KUKA KRL program: Reset_CT.src, Reset_CT.dat

--- Reset_CT.src ---
&ACCESS RVP
&REL 1
DEF  Reset_CT ( )
   ;FOLD INI;%{PE}
      ;FOLD BASISTECH INI
         GLOBAL INTERRUPT DECL 3 WHEN $STOPMESS==TRUE DO IR_STOPM ( )
         INTERRUPT ON 3
         BAS (#INITMOV,0 )
      ;ENDFOLD (BASISTECH INI)
      ;FOLD USER INI
         ;Make your modifications here

      ;ENDFOLD (USER INI)
   ;ENDFOLD (INI)

;Pone a 0 contadore de tiempo de ciclo

;Control Tiempo de ciclo
ALT_TC=1
POS_BAT_TC=1
INDICE_RACK=1
INDICE_PICK=1
INDICE_DROP=1
INDICE_ARRAYS_CPB=1
INDICE_ARRAYS_CPS=1

TC_PICK_RACK1[1]=0
TC_PICK_RACK1[2]=0
TC_PICK_RACK1[3]=0
TC_PICK_RACK1[4]=0
TC_PICK_RACK1[5]=0
TC_PICK_RACK1[6]=0
TC_PICK_RACK1[7]=0
TC_PICK_RACK1[8]=0
TC_PICK_RACK1[9]=0
TC_PICK_RACK1[10]=0
TC_PICK_RACK1[11]=0
TC_PICK_RACK1[12]=0
TC_PICK_RACK1[13]=0
TC_PICK_RACK1[14]=0
TC_PICK_RACK1[15]=0
TC_PICK_RACK1[16]=0
TC_PICK_RACK1[17]=0
TC_PICK_RACK1[18]=0
TC_PICK_RACK1[19]=0
TC_PICK_RACK1[20]=0
TC_PICK_RACK1[21]=0
TC_PICK_RACK1[22]=0
TC_PICK_RACK1[23]=0
TC_PICK_RACK1[24]=0
TC_PICK_RACK1[25]=0
TC_PICK_RACK1[26]=0
TC_PICK_RACK1[27]=0
TC_PICK_RACK1[28]=0
TC_PICK_RACK1[29]=0
TC_PICK_RACK1[30]=0
TC_PICK_RACK1[31]=0
TC_PICK_RACK1[32]=0
TC_PICK_RACK1[33]=0
TC_PICK_RACK1[34]=0
TC_PICK_RACK1[35]=0
TC_PICK_RACK1[36]=0

TC_PICK_RACK2[1]=0
TC_PICK_RACK2[2]=0
TC_PICK_RACK2[3]=0
TC_PICK_RACK2[4]=0
TC_PICK_RACK2[5]=0
TC_PICK_RACK2[6]=0
TC_PICK_RACK2[7]=0
TC_PICK_RACK2[8]=0
TC_PICK_RACK2[9]=0
TC_PICK_RACK2[10]=0
TC_PICK_RACK2[11]=0
TC_PICK_RACK2[12]=0
TC_PICK_RACK2[13]=0
TC_PICK_RACK2[14]=0
TC_PICK_RACK2[15]=0
TC_PICK_RACK2[16]=0
TC_PICK_RACK2[17]=0
TC_PICK_RACK2[18]=0
TC_PICK_RACK2[19]=0
TC_PICK_RACK2[20]=0
TC_PICK_RACK2[21]=0
TC_PICK_RACK2[22]=0
TC_PICK_RACK2[23]=0
TC_PICK_RACK2[24]=0
TC_PICK_RACK2[25]=0
TC_PICK_RACK2[26]=0
TC_PICK_RACK2[27]=0
TC_PICK_RACK2[28]=0
TC_PICK_RACK2[29]=0
TC_PICK_RACK2[30]=0
TC_PICK_RACK2[31]=0
TC_PICK_RACK2[32]=0
TC_PICK_RACK2[33]=0
TC_PICK_RACK2[34]=0
TC_PICK_RACK2[35]=0
TC_PICK_RACK2[36]=0

TC_CARTON[1]=0
TC_CARTON[2]=0
TC_CARTON[3]=0
TC_CARTON[4]=0

TC_DROP[1]=0
TC_DROP[2]=0
TC_DROP[3]=0
TC_DROP[4]=0

TC_CP_BIG[1]=0
TC_CP_BIG[2]=0
TC_CP_BIG[3]=0

TC_CP_SMALL[1]=0
TC_CP_SMALL[2]=0
TC_CP_SMALL[3]=0
TC_CP_SMALL[4]=0
TC_CP_SMALL[5]=0
TC_CP_SMALL[6]=0
TC_CP_SMALL[7]=0
TC_CP_SMALL[8]=0
TC_CP_SMALL[9]=0

TC_ARRAY_CPB[1]=0
TC_ARRAY_CPB[2]=0
TC_ARRAY_CPB[3]=0
TC_ARRAY_CPB[4]=0
TC_ARRAY_CPB[5]=0
TC_ARRAY_CPB[6]=0
TC_ARRAY_CPB[7]=0
TC_ARRAY_CPB[8]=0
TC_ARRAY_CPB[9]=0
TC_ARRAY_CPB[10]=0
TC_ARRAY_CPB[11]=0
TC_ARRAY_CPB[12]=0
TC_ARRAY_CPB[13]=0
TC_ARRAY_CPB[14]=0
TC_ARRAY_CPB[15]=0
TC_ARRAY_CPB[16]=0
TC_ARRAY_CPB[17]=0
TC_ARRAY_CPB[18]=0

END

--- Reset_CT.dat ---
&ACCESS RVP
&REL 1
DEFDAT  Reset_CT
;FOLD EXTERNAL DECLARATIONS;%{PE}%MKUKATPBASIS,%CEXT,%VCOMMON,%P
;FOLD BASISTECH EXT;%{PE}%MKUKATPBASIS,%CEXT,%VEXT,%P
EXT  BAS (BAS_COMMAND  :IN,REAL  :IN )
;ENDFOLD (BASISTECH EXT)
;FOLD USER EXT;%{E}%MKUKATPUSER,%CEXT,%VEXT,%P
;Make your modifications here

;ENDFOLD (USER EXT)
;ENDFOLD (EXTERNAL DECLARATIONS)
ENDDAT
